// TwinCAT 3 PLC project EtherCAT_Test_1
// ProgramVersion: 3.1.4023.0
// libraries:
//   Tc2_EtherCAT, * (Beckhoff Automation GmbH)
//   Tc2_HVAC, * (Beckhoff Automation GmbH)
//   Tc2_Standard, * (Beckhoff Automation GmbH)
//   Tc2_System, * (Beckhoff Automation GmbH)
//   Tc3_Module, * (Beckhoff Automation GmbH)
// project tree:
//   DUTs/ ST_TypeOfPositioning.TcDUT
//   GVLs/ GVL.TcGVL
//   / PlcTask.TcTTO
//   POUs/ MAIN.TcPOU, P_ProfilePositionModeTest.TcPOU, P_VelocityModeTest.TcPOU, StartUpTests.TcPOU, ST_PlcErrorStartUp.TcDUT
//   POUs/ProfilePositionMode/ FB_EnableDevice.TcPOU, Motion.TcPOU
//   POUs/VelocityMode/ BasicTests.TcPOU, VelocityMode.TcPOU

CONFIGURATION EtherCAT_Test_1
    RESOURCE PLC ON TwinCAT3
        TASK PlcTask(INTERVAL := T#10ms, PRIORITY := 20);
        PROGRAM MAIN WITH PlcTask : MAIN;
    END_RESOURCE
END_CONFIGURATION

// ---- DUTs/ST_TypeOfPositioning.TcDUT
TYPE ST_TypeOfPositioning :
STRUCT
	bStartImmediately			: BOOL; (*if Bool is true, target position is absolute, otherwise relative*)
	bAbsolutePositioning		: BOOL; (*if Bool is true, velocity does not change, when first target position is reached - no braking*)
	bChangeOnSetPoint			: BOOL; (*if set true, moving command is executed immediately*)
	nReferencing				: BYTE;
	(*describes positioning behaviour 
		- 1: Positioning relative to previous target position
		- 2: Positioning relative to default value of ramp generator
		- 3: Positioning relative to actual position*)	
END_STRUCT
END_TYPE

// ---- POUs/ST_PlcErrorStartUp.TcDUT
TYPE ST_PlcErrorStartUp :
STRUCT
	bPlcError		: BOOL;
	bErrorCode		: ARRAY[1..4] OF UDINT;
END_STRUCT
END_TYPE

// ---- GVLs/GVL.TcGVL
{attribute 'qualified_only'}
VAR_GLOBAL
	sNetId				: T_AmsNetId := '5.109.65.175.2.1';
	nSlaveAddr			: UINT := 1004;
	
	Controlword AT%Q*		: UINT;	
	Statusword AT%I*		: UINT;
	
	bReset					: BOOL;
END_VAR

// ---- POUs/MAIN.TcPOU
PROGRAM MAIN
VAR_INPUT
	Controlword AT%Q*		: UINT;	
	TargetPosition AT%Q*	: DINT;
END_VAR
VAR_OUTPUT
	Statusword AT%I*		: UINT;
END_VAR

VAR
	bStartUpTest			: BOOL;
	bVelocityModeActive		: BOOL := FALSE;
END_VAR	

VAR
	aTemperatureObjects		: ARRAY[1..2] OF INT := [1,1]; 	//0x2200, 0x2202
	aMOPObjects				: ARRAY[1..2] OF INT := [1,1]; 	//0x6060, 0x6061
	aControlStatusWords		: ARRAY[1..2] OF INT := [1,1]; 	//0x6040, 0x6041
	bTargetPosition			: BOOL;							//0x607A
	
	fbSetToPPMode			: FB_EcCoeSdoWrite;
	fbSetToVelocityMode		: FB_EcCoeSdoWrite;
	bSetToPPMode			: BOOL;
	bSetToVelocityMode		: BOOL := TRUE;
	tSetToPPMode			: TON;
	fSetToVelocityMode		: F_TRIG;
	nModeOfOperation		: UDINT := 2;
	bBasicTest 				: BOOL := FALSE;
END_VAR

//StartUpTests(bTrigger := bStartUpTest,
//	aTemperatureObjects := aTemperatureObjects,
//	aControlStatusWords := aControlStatusWords,
//	aMOPObjects := aMOPObjects,
//	sNetID := GVL.sNetId,
//	nSlaveAddr := GVL.nSlaveAddr);
(*
fbSetToPPMode(sNetId := GVL.sNetId, 
				nSlaveAddr := GVL.nSlaveAddr,
				nIndex := 16#6060,
				pSrcBuf := ADR(nModeOfOperation),
				cbBufLen := SIZEOF (nModeOfOperation),
				bExecute := bSetToPPMode);
tSetToPPMode(IN := bSetToPPMode,
				PT := T#250MS);
bSetToPPMode := TRUE;
IF tSetToPPMode.Q THEN
	P_ProfilePositionModeTest();	
END_IF
*)
IF bBasicTest THEN
	BasicTests();
ELSE
//TODO read IF velocitymode was set via FB
fbSetToVelocityMode(sNetId := GVL.sNetId, 
				nSlaveAddr := GVL.nSlaveAddr,
				nIndex := 16#6060,
				pSrcBuf := ADR(nModeOfOperation),
				cbBufLen := SIZEOF (nModeOfOperation),
				bExecute := bSetToVelocityMode);
fSetToVelocityMode(CLK := fbSetToVelocityMode.bBusy);

IF fSetToVelocityMode.Q THEN
	bVelocityModeActive := TRUE;
	ADSLOGSTR(msgCtrlMask := ADSLOG_MSGTYPE_HINT,
				msgFmtStr := 'Set to velocity mode.',
				strArg := '');
END_IF
IF bVelocityModeActive THEN
	P_VelocityModeTest();
END_IF
END_IF

END_PROGRAM

// ---- POUs/VelocityMode/BasicTests.TcPOU
PROGRAM BasicTests
VAR
	bSetVelocity			: BOOL;
	bStop					: BOOL;
	nTargetVelocity 		: DINT := 1000;
	fbGetStatusword			: FB_EcCoeSdoRead;
	fbSetVelocityWindow 	: FB_EcCoeSdoWrite;
	fbSetVelocityWindowTime	: FB_EcCoeSdoWrite;
	fbProfileVelocityMode 	: ProfileVelocityMode;
	nStatusWord				: DINT;
	bGetStatusword			: BOOL;
	tGetStatusword: TON;
	bTargetReached: BOOL;
	bSpeedIsZero: BOOL;
	nVelocityWindow		: DINT := 50;
	bSetVelocityWindow: BOOL;
	nVelocityWindowTime: DINT := 100;
END_VAR


fbProfileVelocityMode(sNetID := GVL.sNetId,
					nSlaveAddr := GVL.nSlaveAddr,
					nTargetVelocity := nTargetVelocity,
					bSetVelocity := bSetVelocity);	
			
IF bStop THEN
	MAIN.Controlword := 0;
	GVL.bReset := TRUE;
	bStop := FALSE;
END_IF

tGetStatusword(IN := bGetStatusword,
					PT := T#50MS);	
IF tGetStatusword.Q THEN
	bGetStatusword := FALSE;
ELSE
	bGetStatusword := TRUE;		
END_IF
// set parameter
fbSetVelocityWindow(sNetId := GVL.sNetId,
						nSlaveAddr := GVL.nSlaveAddr,
						nIndex := 16#606D,
						nSubindex := 0,
						pSrcBuf := ADR(nVelocityWindow),
						cbBufLen := SIZEOF(nVelocityWindow),
						bExecute := bSetVelocityWindow);
fbSetVelocityWindow(sNetId := GVL.sNetId,
						nSlaveAddr := GVL.nSlaveAddr,
						nIndex := 16#606F,
						nSubindex := 0,
						pSrcBuf := ADR(nVelocityWindow),
						cbBufLen := SIZEOF(nVelocityWindow),
						bExecute := bSetVelocityWindow);
						
fbSetVelocityWindowTime(sNetId := GVL.sNetId,
						nSlaveAddr := GVL.nSlaveAddr,
						nIndex := 16#606E,
						nSubindex := 0,
						pSrcBuf := ADR(nVelocityWindowTime),
						cbBufLen := SIZEOF(nVelocityWindowTime),
						bExecute := bSetVelocityWindow);
fbSetVelocityWindowTime(sNetId := GVL.sNetId,
						nSlaveAddr := GVL.nSlaveAddr,
						nIndex := 16#6070,
						nSubindex := 0,
						pSrcBuf := ADR(nVelocityWindowTime),
						cbBufLen := SIZEOF(nVelocityWindowTime),
						bExecute := bSetVelocityWindow);
//end set parameters

fbGetStatusword(sNetId := GVL.sNetId,
				nSlaveAddr := GVL.nSlaveAddr,
				nIndex := 16#6041,
				nSubindex := 0,
				pDstBuf := ADR(nStatusWord),
				cbBufLen := SIZEOF(nStatusWord),
				bExecute := bGetStatusword);
				
IF nStatusWord.10 THEN
	bTargetReached := TRUE;
ELSE
	bTargetReached := FALSE;
END_IF				
IF nStatusWord.12 THEN
	bSpeedIsZero := TRUE;
ELSE
	bSpeedIsZero := FALSE;
END_IF

END_PROGRAM

// ---- POUs/P_VelocityModeTest.TcPOU
PROGRAM P_VelocityModeTest
//general handling
VAR
	bStartTestOfNewDrive			: BOOL;//starts new test
	bRestartTest					: BOOL;//restart if single test failed
	bManuallyRestoreDefaultValues	: BOOL;
	bError							: BOOL := FALSE;//Error handling
	bAckError						: BOOL;//Error handling
	bStopMotor						: BOOL;//Error handling
	bOnFirstIn						: BOOL := TRUE;
END_VAR

//test case success indication variables
VAR
	bSingleTestFailed					: BOOL := FALSE;
	
	bObject6042tested				: BOOL := FALSE;//test case success indication variables
	bObject6043tested				: BOOL := FALSE;//test case success indication variables
	bObject6046tested				: BOOL := FALSE;//test case success indication variables
	bObject6048tested				: BOOL := FALSE;//test case success indication variables
	bObject6049tested				: BOOL := FALSE;//test case success indication variables
	
	bTestBasicOperation_Success		: BOOL := FALSE;//test case success indication variables
	bTestAccel_Success				: BOOL := FALSE;//test case success indication variables	
	bTestDecel_Success				: BOOL := FALSE;//test case success indication variables
	bTestLimits_Success				: BOOL := FALSE;//test case success indication variables
	
	bTestBasicOperation_Failed		: BOOL := FALSE;
	bTestAccel_Failed				: BOOL := FALSE;
	bTestDecel_Failed				: BOOL := FALSE;
	bTestLimits_Failed				: BOOL := FALSE;
	
	bMaxLimitTest_Success			: BOOL := FALSE; //helper for limit
	bMinLimitTest_Success			: BOOL := FALSE; //helper for limit
	bMaxLimitTest_Failed			: BOOL := FALSE; //helper for limit
	bMinLimitTest_Failed			: BOOL := FALSE; //helper for limit	
END_VAR

//relevant parameters for test options
VAR
	fToleranceLimit					: REAL := 0.2; // 20% tolerance
	fToleranceAccDec				: REAL := 0.1; // 10% tolerance
	fToleranceBasicOp				: REAL := 0.02; // 2% tolerance
	nDeltaSpeedRef					: DINT := 300; //speed reference for acc/dec
	nDeltaTimeRef					: DINT := 1; //time reference for acc/dec
	nMinLimitRef					: DINT := 200; //testing this minimum velocity limit
	nMaxLimitRef					: DINT := 1000; //testing this maximum velocity limit	
END_VAR

// default values will be deliberately changed. Persistent variables keep their values also at shutdown of PLC, see https://infosys.beckhoff.com/index.php?content=../content/1031/tc3_plc_intro/2526557579.html&id=
// pressing "restart in run modus" will NOT clear these values!
VAR PERSISTENT
	nDefaultAccSpeed				: DINT;
	nDefaultDecSpeed				: DINT;
	nDefaultAccTime					: DINT;
	nDefaultDecTime					: DINT;
	nDefaultVelocityMinLimit		: DINT;
	nDefaultVelocityMaxLimit		: DINT;
END_VAR

// all variables
VAR	
	eTestMode	: (WAIT_FOR_TEST, READ_DEFAULT_VALUES, WRITE_DEFAULT_VALUES, ERROR, STOP_DRIVE, BASIC_OPERATION, TEST_ACCEL, TEST_DECEL, TEST_LIMITS); 
	step							: INT := 1;
	stepTestMode					: INT := 0; //start in idle mode
	
	bSetControlWord					: BOOL := TRUE;
	fbVelocityMode					: VelocityMode;
	fbGetStatusword					: FB_EcCoeSdoRead;
	fbGetActualVelocity				: FB_EcCoeSdoRead;
//	fbGetVelocityLimitMax			: FB_EcCoeSdoRead;
//	fbGetVelocityLimitMin			: FB_EcCoeSdoRead;
	fbReadVelocityLimits1			: FB_EcCoeSdoRead;
	fbReadVelocityLimits2			: FB_EcCoeSdoRead;
	fbWriteVelocityLimits1			: FB_EcCoESdoWrite;
	fbWriteVelocityLimits2			: FB_EcCoESdoWrite;
	fbWriteAcc1						: FB_EcCoESdoWrite;
	fbWriteAcc2						: FB_EcCoESdoWrite;
	fbReadAcc1						: FB_EcCoeSdoRead;
	fbReadAcc2						: FB_EcCoeSdoRead;
	fbWriteDec1						: FB_EcCoESdoWrite;
	fbWriteDec2						: FB_EcCoESdoWrite;
	fbReadDec1						: FB_EcCoeSdoRead;
	fbReadDec2						: FB_EcCoeSdoRead;
	fbGetVelocityDemand				: FB_EcCoESdoRead;
	fbGetTargetVelocity				: FB_EcCoESdoRead;
	nTargetVelocity					: DINT := 50; //rpm
	nActualVelocity					: DINT;
	nStatusword						: UINT;
	nSpeed							: DINT;
	nTime							: DINT;
		
	bGetCurrentVelocity				: BOOL;
	bGetStatusword					: BOOL;
	bSetVelocity					: BOOL; 
	nTargetVelocityAfterLimit		: DINT;
	tTimeDec1						: TIME;
	tTimeDec2						: TIME;
	nAccMeasured					: REAL;
	nDecMeasured					: REAL;
	bIsAccelerating					: BOOL;
	bIsDecelerating					: BOOL;
	
	bDone							: BOOL;
	nDeltaVelocityTarget			: REAL;
	fDesiredAcceleration			: REAL;
	nVelocityDemand					: DINT;
	nVelocityMinLimit 				: DINT;
	nVelocityMaxLimit 				: DINT;
	bWriteDefaultValues				: BOOL;
	nDecVelocity					: DINT;
	fDesiredDeceleration			: REAL;
	bStopAfterLimitTest				: BOOL;

	tTimeout						: TON;
	tTimer							: TON;
	tGetStatusword					: TON;
	tWaitForCurrentVelocity			: TON;
	tTimeAcc1						: TIME;
	tTimeAcc2						: TIME;
	tDiff							: TIME;
	fTrigger						: F_TRIG;
	fFlag 							: F_TRIG;
	fFlag2 							: F_TRIG;	
	ShowLimitVelocity				: DINT;
END_VAR

IF bTestBasicOperation_Failed OR bTestAccel_Failed OR bTestDecel_Failed OR bMinLimitTest_Failed OR bMaxLimitTest_Failed OR bTestLimits_Failed THEN
	bSingleTestFailed := TRUE;
ELSE bSingleTestFailed := FALSE;
END_IF


tWaitForCurrentVelocity(IN := bGetCurrentVelocity,
							PT := T#10MS);
tGetStatusword(IN := bGetStatusword,
					PT := T#500MS);	
							
IF tWaitForCurrentVelocity.Q THEN
	bGetCurrentVelocity := FALSE;
ELSE
	bGetCurrentVelocity := TRUE;		
END_IF
// read FBs
fbGetStatusword(sNetId := GVL.sNetId,
				nSlaveAddr := GVL.nSlaveAddr,
				nIndex := 16#6041,
				nSubindex := 0,
				pDstBuf := ADR(nStatusWord),
				cbBufLen := SIZEOF(nStatusWord),
				bExecute := bGetStatusword);
				
fbGetActualVelocity(sNetId := GVL.sNetId,
					nSlaveAddr := GVL.nSlaveAddr,
					nIndex := 16#6044,
					nSubindex := 0,
					pDstBuf := ADR(nActualVelocity),
					cbBufLen := SIZEOF(nActualVelocity),
					bExecute := bGetCurrentVelocity);

//write to motor
MAIN.Controlword.4 := bSetControlWord; //velocity demand value shall equal to ramp output value
MAIN.Controlword.5 := bSetControlWord; //ramp output value shall follow ramp input value
MAIN.Controlword.6 := bSetControlWord; //ramp input value shall accord with ramp reference

			
//stop
IF bStopMotor THEN
	MAIN.Controlword := 0;
	stepTestMode := 0;
END_IF


(*TEST SUITE*)	
//error detection
IF bError THEN
	MAIN.Controlword := 0;
	stepTestMode := 0;
	eTestMode := ERROR;
END_IF
// restore stored default values
IF bManuallyRestoreDefaultValues THEN
	bError := FALSE;
	stepTestMode := 0;
	eTestMode := WRITE_DEFAULT_VALUES;
END_IF

CASE eTestMode OF
	WAIT_FOR_TEST:
		tTimeout(IN := FALSE);
		step := 1; //resetting general step counter for use within TestModes
		CASE stepTestMode OF
			0: //idle
				IF bRestartTest THEN //restart inside a test procedure
					GVL.bReset := TRUE;
					bRestartTest := FALSE; 
					bSetControlWord := TRUE;
					bTestBasicOperation_Failed := bTestAccel_Failed := bTestDecel_Failed := bMinLimitTest_Failed := bMaxLimitTest_Failed := bTestLimits_Failed := FALSE;
					stepTestMode := stepTestMode+1;
				END_IF
				IF bStartTestOfNewDrive THEN //start test of a new drive 
					GVL.bReset := TRUE;
					Reset();
					bSetControlWord := TRUE;
					bStartTestOfNewDrive := FALSE;
					eTestMode := READ_DEFAULT_VALUES;
				END_IF
		
			1: 
				IF bTestBasicOperation_Success THEN 
					stepTestMode := stepTestMode+1; 
					bObject6043tested := TRUE;
				ELSE 
					eTestMode := BASIC_OPERATION; 
					ADSLOGSTR(msgCtrlMask := ADSLOG_MSGTYPE_HINT, msgFmtStr := 'Testing basic operation...', strArg := '');
				END_IF 				
			2: 				
				IF bTestAccel_Success THEN 
					stepTestMode := stepTestMode+1; 
					bObject6048tested := TRUE;
				ELSIF nActualVelocity = 0 THEN 
					eTestMode := TEST_ACCEL; 
					bSetControlWord := TRUE; 
					ADSLOGSTR(msgCtrlMask := ADSLOG_MSGTYPE_HINT, msgFmtStr := 'Testing acceleration...', strArg := '');
				END_IF 				
			3: 
				IF bTestDecel_Success THEN 
					stepTestMode := stepTestMode+1; 
					bObject6049tested := TRUE;
				ELSE 
					eTestMode := TEST_DECEL; 
					ADSLOGSTR(msgCtrlMask := ADSLOG_MSGTYPE_HINT, msgFmtStr := 'Testing deceleration...', strArg := '');
				END_IF
			4: 
				IF bTestLimits_Success THEN 
					stepTestMode := stepTestMode+1; 
					bObject6046tested := TRUE;
				ELSE 
					eTestMode := TEST_LIMITS; 
					ADSLOGSTR(msgCtrlMask := ADSLOG_MSGTYPE_HINT, msgFmtStr := 'Testing limits...', strArg := '');
				END_IF				
			
			5: //all tests successful
				MAIN.Controlword := 0;
				ADSLOGSTR(msgCtrlMask := ADSLOG_MSGTYPE_HINT, msgFmtStr := 'All tests successful!', strArg := '');
				stepTestMode := 0; //idle
		END_CASE	
	
		
	(* Error handling *)
	ERROR:
		MAIN.Controlword := 0;
		bSetControlWord := FALSE;
		step := 1;
		IF bAckError OR bRestartTest THEN
			bAckError := FALSE;
			bError := FALSE;
			
			eTestMode := WAIT_FOR_TEST;
			stepTestMode := 0;
		END_IF


	READ_DEFAULT_VALUES: 
		CASE step OF
			1: //read acc
				ReadAcc(nDeltaSpeed := nDefaultAccSpeed, nDeltaTime := nDefaultAccTime, bDone => bDone);
				IF bDone THEN
					step := step+1;
				END_IF
			2: //read dec
				ReadDec(nDeltaSpeed := nDefaultDecSpeed, nDeltaTime := nDefaultDecTime, bDone => bDone);
				IF bDone THEN
					step := step+1;
				END_IF				
			3: //read limits
				ReadVelocityLimits(nVelocityMinLimit := nDefaultVelocityMinLimit, nVelocityMaxLimit := nDefaultVelocityMaxLimit, bDone => bDone);
				IF bDone THEN
					step := step+1;
				END_IF
			4: 
				eTestMode := WAIT_FOR_TEST;			
				ADSLOGSTR(msgCtrlMask := ADSLOG_MSGTYPE_HINT, msgFmtStr := 'Default values read.', strArg := '');
				stepTestMode := 1; //start test basic operation
		END_CASE
		
		
	WRITE_DEFAULT_VALUES: 
		IF bOnFirstIn THEN 
			step := 1;
		END_IF
		CASE step OF
			1: //write acc
				bOnFirstIn := FALSE;
				WriteAcc(nDeltaSpeedRef := nDefaultAccSpeed, nDeltaTimeRef := nDefaultAccTime, bDone => bDone);
				IF bDone THEN
					step := step+1;
				END_IF
			2: 
				ReadAcc(nDeltaSpeed := nSpeed, nDeltaTime := nTime, bDone => bDone);
				IF nSpeed = nDefaultAccSpeed AND nTime = nDefaultAccTime AND bDone THEN
					step := step+1;
				END_IF
			3: //write dec
				WriteDec(nDeltaSpeedRef := nDefaultDecSpeed, nDeltaTimeRef := nDefaultDecTime, bDone => bDone);
				IF bDone THEN
					step := step+1;
				END_IF	
			4:
				ReadDec(nDeltaSpeed := nSpeed, nDeltaTime := nTime, bDone => bDone);
				IF nSpeed = nDefaultDecSpeed AND nTime = nDefaultDecTime AND bDone THEN
					step := step+1;
				END_IF
			
			5: //write limits
				WriteVelocityLimits(nVelocityMinLimit := nDefaultVelocityMinLimit, nVelocityMaxLimit := nDefaultVelocityMaxLimit, bDone => bDone);
				IF bDone THEN
					step := step+1;
				END_IF
			6: 
				ReadVelocityLimits(nVelocityMinLimit := nVelocityMinLimit, nVelocityMaxLimit := nVelocityMaxLimit, bDone => bDone);
				IF nVelocityMinLimit = nDefaultVelocityMinLimit AND nVelocityMaxLimit = nDefaultVelocityMaxLimit AND bDone THEN
					step := step+1;
				END_IF

			7: 
				eTestMode := WAIT_FOR_TEST;	
				ADSLOGSTR(msgCtrlMask := ADSLOG_MSGTYPE_HINT,
					msgFmtStr := 'Default values restored. Acc, dec and limits',
					strArg := '');		
				IF bSingleTestFailed THEN
					bError := TRUE;
				END_IF
				IF bStopAfterLimitTest THEN
					bStopAfterLimitTest := FALSE;
					eTestMode := STOP_DRIVE;
				END_IF
				bManuallyRestoreDefaultValues := FALSE;
				bOnFirstIn := TRUE;
		END_CASE
		
		
	STOP_DRIVE:
		step := 1;
		nTargetVelocity := 0;
		tTimeout(IN := TRUE, PT := T#15S);
		bSetVelocity := TRUE;
		fbVelocityMode(sNetID := GVL.sNetId,
					nSlaveAddr := GVL.nSlaveAddr,
					nTargetVelocity := nTargetVelocity,
					bSetVelocity := bSetVelocity,
					nTargetVelocityAfterLimit => nTargetVelocityAfterLimit);
		IF nActualVelocity = 0 THEN
			IF bWriteDefaultValues THEN
				bWriteDefaultValues := FALSE;
				eTestMode := WRITE_DEFAULT_VALUES;
			ELSE
				eTestMode := WAIT_FOR_TEST;
			END_IF
		END_IF
		
		IF tTimeout.Q THEN
			bError := TRUE;
			ADSLOGSTR(msgCtrlMask := ADSLOG_MSGTYPE_HINT,
				msgFmtStr := 'Timeout when shutting down drive. Please restore default values manually.',
				strArg := '');
		END_IF
	
	(* Test basic operation *)
	BASIC_OPERATION:
		tTimeout(IN := TRUE, PT := T#10S);
		CASE step OF
		1:	
			nTargetVelocity := 300; //rpm
			bSetVelocity := TRUE;
			fbVelocityMode(sNetID := GVL.sNetId,
						nSlaveAddr := GVL.nSlaveAddr,
						nTargetVelocity := nTargetVelocity,
						bSetVelocity := bSetVelocity,
						nTargetVelocityAfterLimit => nTargetVelocityAfterLimit);
			IF NOT fbVelocityMode.bBusy THEN //now velocity is set
				step := step+1;
			END_IF				
		2: 
			fbGetTargetVelocity(sNetId := GVL.sNetId,
				nSlaveAddr := GVL.nSlaveAddr,
				nIndex := 16#6042,
				nSubIndex := 0,
				pDstBuf := ADR(nVelocityDemand),
				cbBufLen := SIZEOF(nVelocityDemand),
				bExecute := TRUE);
			fFlag(CLK := fbGetTargetVelocity.bBusy);
			IF fFlag.Q AND nVelocityDemand = nTargetVelocity THEN
				fbGetTargetVelocity(bExecute := FALSE);
				bObject6042tested := TRUE;
				step := step+1;
			END_IF		
		3:  
			tTimer(IN:=TRUE, PT:=T#3S);
			IF tTimer.Q THEN
				tTimer(IN:=FALSE);
				step := step+1;
			END_IF
		4:
			IF  TO_REAL(nActualVelocity) > ((1-fToleranceBasicOp)*TO_REAL(nTargetVelocityAfterLimit)) 
			AND TO_REAL(nActualVelocity) < ((1+fToleranceBasicOp)*TO_REAL(nTargetVelocityAfterLimit)) THEN // Vsoll = Vist with 2% tolerance
				fbGetVelocityDemand(sNetId := GVL.sNetId,
					nSlaveAddr := GVL.nSlaveAddr,
					nIndex := 16#6043,
					nSubIndex := 0,
					pDstBuf := ADR(nVelocityDemand),
					cbBufLen := SIZEOF(nVelocityDemand),
					bExecute := TRUE);
				fFlag2(CLK := fbGetVelocityDemand.bBusy);
				
				IF fFlag2.Q THEN
					fbGetVelocityDemand(bExecute := FALSE);
					IF nVelocityDemand = nTargetVelocity THEN
						bTestBasicOperation_Success := TRUE; //set success indication	
						step := step+1;								
						ADSLOGSTR(msgCtrlMask := ADSLOG_MSGTYPE_HINT,
							msgFmtStr := 'Basic operation test success.',
							strArg := '');
					END_IF
				END_IF
			ELSIF nActualVelocity > 2*nTargetVelocityAfterLimit THEN
				bError := TRUE;
				bTestBasicOperation_Failed := TRUE;
			END_IF				
			
		5:	//soft stop motor
			eTestMode := STOP_DRIVE;			
		END_CASE
		
		//Error handling in wait_for_test
		IF tTimeout.Q THEN
			bTestBasicOperation_Failed := TRUE;
			bError := TRUE;
			ADSLOGSTR(msgCtrlMask := ADSLOG_MSGTYPE_HINT,
				msgFmtStr := 'Basic operation test failed. Timeout.',
				strArg := '');
		END_IF

	
	(* Test acceleration target *)
	TEST_ACCEL:
		tTimeout(IN := TRUE, PT := T#10S); 
		CASE step OF
			1: //set acceleration values
				WriteAcc(nDeltaSpeedRef := nDeltaSpeedRef, nDeltaTimeRef := nDeltaTimeRef, bDone => bDone);
				IF bDone THEN
					step := step+1;
				END_IF
				
			2: //read acceleration
				ReadAcc(nDeltaSpeed := nSpeed, nDeltaTime := nTime, bDone => bDone); 
				IF nSpeed = nDeltaSpeedRef AND nTime = nDeltaTimeRef AND bDone THEN //Acceleration values were set correctly
					step := step+1;
				END_IF
				
			3: //set drive to TargetVelocity and measure acceleration time
				nTargetVelocity := 2000;
				nDeltaVelocityTarget := 0.995*TO_REAL(nTargetVelocity); //needs to be a little lower than target due to acc ramping
				fDesiredAcceleration := TO_REAL(nDeltaSpeedRef/nDeltaTimeRef); // acc reference
				
				bSetVelocity := TRUE;
				fbVelocityMode(sNetID := GVL.sNetId,
							nSlaveAddr := GVL.nSlaveAddr,
							nTargetVelocity := nTargetVelocity,
							bSetVelocity := bSetVelocity,
							nTargetVelocityAfterLimit => nTargetVelocityAfterLimit);
				fTrigger(CLK := fbVelocityMode.bBusy);
				IF fTrigger.Q THEN
					tTimeAcc1 := TIME();
					step := step+1;
				END_IF
			
			4:
				tTimer(IN:=TRUE, PT:=T#50MS);
				IF tTimer.Q THEN
					tTimer(IN:=FALSE);
					step := step+1;
				END_IF
				
			5:
				IF TO_REAL(nActualVelocity) >= nDeltaVelocityTarget THEN 
					tTimeAcc2 := TIME();
					tDiff := tTimeAcc2 - tTimeAcc1; //time difference of drive to reach nSpeedRef
					nAccMeasured := TO_REAL(nActualVelocity*1000/TIME_TO_DINT(tDiff)); //time in ms
					step := step+1;
				END_IF

			6: //validate result
				IF  nAccMeasured > ((1-fToleranceAccDec)*fDesiredAcceleration) 
				AND nAccMeasured < ((1+fToleranceAccDec)*fDesiredAcceleration) THEN //within range of tolerance: default 10%
					bTestAccel_Success := TRUE;
					ADSLOGSTR(msgCtrlMask := ADSLOG_MSGTYPE_HINT,
					msgFmtStr := 'Acceleration test success.',
					strArg := '');
				ELSE
					bTestAccel_Failed := TRUE;
					ADSLOGSTR(msgCtrlMask := ADSLOG_MSGTYPE_HINT,
						msgFmtStr := 'Acceleration test failed. Motor acceleration not within range of reference values.',
						strArg := '');
				END_IF
				bWriteDefaultValues := TRUE;
				eTestMode := STOP_DRIVE; //stop and restore default variables
		END_CASE
		
		//Error handling timeout
		IF tTimeout.Q THEN
			eTestMode := WRITE_DEFAULT_VALUES; //restore default variables
			bTestAccel_Failed := TRUE;
			ADSLOGSTR(msgCtrlMask := ADSLOG_MSGTYPE_HINT,
				msgFmtStr := 'Acceleration test failed. Timeout.',
				strArg := '');
		END_IF
		
	
		
(* Test acceleration target *)
	TEST_DECEL:
		tTimeout(IN := TRUE, PT := T#15S); 
		CASE step OF
			1: //set deceleration values
				WriteDec(nDeltaSpeedRef := nDeltaSpeedRef, nDeltaTimeRef := nDeltaTimeRef, bDone => bDone);
				IF bDone THEN
					step := step+1;
				END_IF
				
			2: //read deceleration
				ReadDec(nDeltaSpeed := nSpeed, nDeltaTime := nTime, bDone => bDone); 
				IF nSpeed = nDeltaSpeedRef AND nTime = nDeltaTimeRef AND bDone THEN //Acceleration values were set correctly
					step := step+1;
				END_IF
				
			3: //set drive to velocity
				nTargetVelocity := 1500;
				nDecVelocity := nTargetVelocity;	
				fDesiredDeceleration := TO_REAL(nDeltaSpeedRef/nDeltaTimeRef); // dec reference		
				bSetVelocity := TRUE;
				fbVelocityMode(sNetID := GVL.sNetId,
							nSlaveAddr := GVL.nSlaveAddr,
							nTargetVelocity := nTargetVelocity,
							bSetVelocity := bSetVelocity,
							nTargetVelocityAfterLimit => nTargetVelocityAfterLimit);
				tTimer(IN:=TRUE, PT:=T#1500MS);
				IF tTimer.Q THEN
					tTimer(IN:=FALSE);
					step := step+1;
				END_IF
			
			4:
				IF nActualVelocity > 0.99*nTargetVelocityAfterLimit THEN 
					nTargetVelocity := 0;
					step := step+1;
				END_IF

			5: //test run of drive for validation of deceleration 
				bSetVelocity := TRUE;
				fbVelocityMode(sNetID := GVL.sNetId,
							nSlaveAddr := GVL.nSlaveAddr,
							nTargetVelocity := nTargetVelocity,
							bSetVelocity := bSetVelocity,
							nTargetVelocityAfterLimit => nTargetVelocityAfterLimit);
				fTrigger(CLK := fbVelocityMode.bBusy);
				IF fTrigger.Q THEN
					tTimeDec1 := TIME();
					step := step+1;
				END_IF
				
			6:
				IF nActualVelocity = nTargetVelocity THEN
					tTimeDec2 := TIME();
					tDiff := tTimeDec2 - tTimeDec1; //time difference of drive to decelerate
					nDecMeasured := TO_REAL(nDecVelocity*1000/TIME_TO_DINT(tDiff));
					step := step+1;
				END_IF
			
			7:	//validation
				IF  nDecMeasured > ((1-fToleranceAccDec)*fDesiredDeceleration) 
				AND nDecMeasured < ((1+fToleranceAccDec)*fDesiredDeceleration) THEN //within range of tolerance: default 10%
					bTestDecel_Success := TRUE;
					ADSLOGSTR(msgCtrlMask := ADSLOG_MSGTYPE_HINT,
					msgFmtStr := 'Deceleration test success.',
					strArg := '');
				ELSE
					bTestDecel_Failed := TRUE;
					ADSLOGSTR(msgCtrlMask := ADSLOG_MSGTYPE_WARN,
						msgFmtStr := 'Deceleration test failed. Motor deceleration not within range of reference values.',
						strArg := '');
				END_IF
				bWriteDefaultValues := TRUE;
				eTestMode := STOP_DRIVE; //stop and restore default variables
		END_CASE
		
		//Error handling timeout
		IF tTimeout.Q THEN
			eTestMode := WRITE_DEFAULT_VALUES; //restore default variables
			bTestDecel_Failed := TRUE;
			ADSLOGSTR(msgCtrlMask := ADSLOG_MSGTYPE_WARN,
				msgFmtStr := 'Deceleration test failed. Timeout.',
				strArg := '');
		END_IF
		

	
//	(* Test velocity limtis *)
	TEST_LIMITS: 
		tTimeout(IN:=TRUE, PT:=T#15S);
		CASE step OF
			1: 
				nTargetVelocity := 2000;
				WriteVelocityLimits(nVelocityMinLimit := nMinLimitRef, nVelocityMaxLimit := nMaxLimitRef, bDone => bDone);
				IF bDone THEN
					step := step+1;
				END_IF
				
			2: //test max limit
				bSetVelocity := TRUE;
				fbVelocityMode(sNetID := GVL.sNetId,
							nSlaveAddr := GVL.nSlaveAddr,
							nTargetVelocity := nTargetVelocity,
							bSetVelocity := bSetVelocity,
							nTargetVelocityAfterLimit => nTargetVelocityAfterLimit);
				IF NOT fbVelocityMode.bBusy THEN
					bIsAccelerating := TRUE;
					step := step+1;
				END_IF
			
			3:
				tTimer(IN := bIsAccelerating, PT := T#3S); //run for x seconds
				IF tTimer.Q THEN 
					tTimer(IN:=FALSE);
					step := step+1;
				END_IF
			
			4:
				IF TO_REAL(nActualVelocity) > ((1+fToleranceLimit)*TO_REAL(nMaxLimitRef))(* 20% overshot accounted *) THEN 
					bMaxLimitTest_Failed := TRUE;
					eTestMode := WRITE_DEFAULT_VALUES;
					ADSLOGSTR(msgCtrlMask := ADSLOG_MSGTYPE_WARN,
						msgFmtStr := 'Max limit test failed.',
						strArg := '');			
				ELSE
					bMaxLimitTest_Success := TRUE;
					ADSLOGSTR(msgCtrlMask := ADSLOG_MSGTYPE_HINT,
						msgFmtStr := 'Max limit test success.',
						strArg := '');
					step := step+1;
				END_IF
				bIsAccelerating := FALSE;
				nTargetVelocity := 0;
				
			5: //test min limit
				bSetVelocity := TRUE;
				fbVelocityMode(sNetID := GVL.sNetId,
							nSlaveAddr := GVL.nSlaveAddr,
							nTargetVelocity := nTargetVelocity,
							bSetVelocity := bSetVelocity,
							nTargetVelocityAfterLimit => nTargetVelocityAfterLimit);
				IF NOT fbVelocityMode.bBusy THEN
					bIsDecelerating := TRUE;
					step := step+1;
				END_IF
								
			6:
				tTimer(IN := bIsDecelerating, PT := T#3S); //run for x seconds
				IF tTimer.Q THEN 
					tTimer(IN:=FALSE);
					step := step+1;
				END_IF
			
			7:
				// a way for dynamic time determination
//				fTimeFaktor := DINT_TO_REAL((nActualVelocity-nTargetVelocity)/nSpeedDec); 
//				tDecTime := REAL_TO_TIME(2000+fTimeFaktor * nDefaultDecTime*1000); //acceleration time, min 2s
//				tTimer(IN := bIsDecelerating, PT := tDecTime);
				IF TO_REAL(nActualVelocity) < ((1-fToleranceLimit)*TO_REAL(nMinLimitRef))(*20% overshot accounted*) THEN 
					bMinLimitTest_Failed := TRUE;
					ADSLOGSTR(msgCtrlMask := ADSLOG_MSGTYPE_WARN,
						msgFmtStr := 'Min limit test failed.',
						strArg := '');										
				ELSE //time at witch the drive would be on targetvelocity without limit acitve
					bMinLimitTest_Success := TRUE;
					ADSLOGSTR(msgCtrlMask := ADSLOG_MSGTYPE_HINT,
						msgFmtStr := 'Min limit test success.',
						strArg := '');
				END_IF
				ShowLimitVelocity := nActualVelocity;
				step := step+1;
				bIsDecelerating := FALSE;
			
			8:
				IF bMinLimitTest_Success AND bMaxLimitTest_Success THEN
					bTestLimits_Success := TRUE;
					ADSLOGSTR(msgCtrlMask := ADSLOG_MSGTYPE_HINT,
						msgFmtStr := 'Limit test success.',
						strArg := '');
				ELSE
					bTestLimits_Failed := TRUE;
				END_IF
				bStopAfterLimitTest := TRUE;
				eTestMode := WRITE_DEFAULT_VALUES; //stop and restore default variables				
		END_CASE

END_CASE

METHOD ReadAcc : BOOL
VAR_IN_OUT
	nDeltaSpeed 	: DINT;
	nDeltaTime 		: DINT;
	//bRead : BOOL;
END_VAR
VAR_OUTPUT
	bDone			: BOOL;
END_VAR
bDone := FALSE;
//IF bRead THEN
	fbReadAcc1(sNetId := GVL.sNetId,
				nSlaveAddr := GVL.nSlaveAddr,
				nIndex := 16#6048,
				nSubindex := 1, //delta speed
				pDstBuf := ADR(nDeltaSpeed),
				cbBufLen := SIZEOF(nDeltaSpeed),
				bExecute := TRUE);
	
	fbReadAcc2(sNetId := GVL.sNetId,
				nSlaveAddr := GVL.nSlaveAddr,
				nIndex := 16#6048,
				nSubindex := 2, //delta time
				pDstBuf := ADR(nDeltaTime),
				cbBufLen := SIZEOF(nDeltaTime),
				bExecute := TRUE);
//END_IF
IF NOT fbReadAcc1.bBusy AND NOT fbReadAcc2.bBusy THEN
	fbReadAcc1(bExecute := FALSE); 
	fbReadAcc2(bExecute := FALSE); 
	//bRead := FALSE;
	bDone := TRUE;
END_IF
END_METHOD

METHOD ReadDec : BOOL
VAR_IN_OUT
	nDeltaSpeed 	: DINT;
	nDeltaTime 		: DINT;
END_VAR
VAR_OUTPUT
	bDone			: BOOL;
END_VAR
bDone := FALSE;
fbReadDec1(sNetId := GVL.sNetId,
			nSlaveAddr := GVL.nSlaveAddr,
			nIndex := 16#6049,
			nSubindex := 1, //delta speed
			pDstBuf := ADR(nDeltaSpeed),
			cbBufLen := SIZEOF(nDeltaSpeed),
			bExecute := TRUE);

fbReadDec2(sNetId := GVL.sNetId,
			nSlaveAddr := GVL.nSlaveAddr,
			nIndex := 16#6049,
			nSubindex := 2, //delta time
			pDstBuf := ADR(nDeltaTime),
			cbBufLen := SIZEOF(nDeltaTime),
			bExecute := TRUE);

IF NOT fbReadDec1.bBusy AND NOT fbReadDec2.bBusy THEN
	fbReadDec1(bExecute := FALSE); 
	fbReadDec2(bExecute := FALSE); 
	bDone := TRUE;
END_IF
END_METHOD

METHOD ReadVelocityLimits : BOOL
VAR_IN_OUT
	nVelocityMinLimit 	: DINT;
	nVelocityMaxLimit 	: DINT;
END_VAR
VAR_OUTPUT
	bDone			: BOOL;
END_VAR
bDone := FALSE;
	fbReadVelocityLimits1(sNetId := GVL.sNetId,
			nSlaveAddr := GVL.nSlaveAddr,
			nIndex := 16#6046,
			nSubindex := 1, //v_min
			pDstBuf := ADR(nVelocityMinLimit),
			cbBufLen := SIZEOF(nVelocityMinLimit),
			bExecute := TRUE);
	
	fbReadVelocityLimits2(sNetId := GVL.sNetId,
			nSlaveAddr := GVL.nSlaveAddr,
			nIndex := 16#6046,
			nSubindex := 2, //v_max
			pDstBuf := ADR(nVelocityMaxLimit),
			cbBufLen := SIZEOF(nVelocityMaxLimit),
			bExecute := TRUE);
			
IF NOT fbReadVelocityLimits1.bBusy AND NOT fbReadVelocityLimits2.bBusy THEN
	fbReadVelocityLimits1(bExecute := FALSE); 
	fbReadVelocityLimits2(bExecute := FALSE); 
	bDone := TRUE;
END_IF
END_METHOD

METHOD Reset : BOOL
VAR_INPUT
END_VAR
bObject6042tested				:= FALSE;
bObject6043tested				:= FALSE;
bObject6046tested				:= FALSE;
bObject6048tested				:= FALSE;
bObject6049tested				:= FALSE;

bTestBasicOperation_Success		:= FALSE;
bTestAccel_Success				:= FALSE;	
bTestDecel_Success				:= FALSE;
bTestLimits_Success				:= FALSE;

bTestBasicOperation_Failed		:= FALSE;
bTestAccel_Failed				:= FALSE;
bTestDecel_Failed				:= FALSE;
bTestLimits_Failed				:= FALSE;
bSingleTestFailed					:= FALSE;

bMaxLimitTest_Success			:= FALSE;
bMinLimitTest_Success			:= FALSE;
bMaxLimitTest_Failed			:= FALSE;
bMinLimitTest_Failed			:= FALSE;
END_METHOD

METHOD WriteAcc : BOOL
VAR_IN_OUT
	nDeltaSpeedRef	: DINT;
	nDeltaTimeRef	: DINT;
END_VAR
VAR_OUTPUT
	bDone 			: BOOL;
END_VAR
bDone := FALSE;
fbWriteAcc1(sNetId := GVL.sNetId,
		nSlaveAddr := GVL.nSlaveAddr,
		nIndex := 16#6048,
		nSubindex := 1, //delta speed
		pSrcBuf := ADR(nDeltaSpeedRef),
		cbBufLen := SIZEOF(nDeltaSpeedRef),
		bExecute := TRUE);	
			
fbWriteAcc2(sNetId := GVL.sNetId,
		nSlaveAddr := GVL.nSlaveAddr,
		nIndex := 16#6048,
		nSubindex := 2, //delta time
		pSrcBuf := ADR(nDeltaTimeRef),
		cbBufLen := SIZEOF(nDeltaTimeRef),
		bExecute := TRUE);

IF NOT fbWriteAcc1.bBusy AND NOT fbWriteAcc2.bBusy THEN
	fbWriteAcc1(bExecute := FALSE); 
	fbWriteAcc2(bExecute := FALSE); 
	bDone := TRUE;
END_IF
END_METHOD

METHOD WriteDec : BOOL
VAR_IN_OUT
	nDeltaSpeedRef	: DINT;
	nDeltaTimeRef	: DINT;
END_VAR
VAR_OUTPUT
	bDone 			: BOOL;
END_VAR
bDone := FALSE;
fbWriteDec1(sNetId := GVL.sNetId,
		nSlaveAddr := GVL.nSlaveAddr,
		nIndex := 16#6049,
		nSubindex := 1, //delta speed
		pSrcBuf := ADR(nDeltaSpeedRef),
		cbBufLen := SIZEOF(nDeltaSpeedRef),
		bExecute := TRUE);	
			
fbWriteDec2(sNetId := GVL.sNetId,
		nSlaveAddr := GVL.nSlaveAddr,
		nIndex := 16#6049,
		nSubindex := 2, //delta time
		pSrcBuf := ADR(nDeltaTimeRef),
		cbBufLen := SIZEOF(nDeltaTimeRef),
		bExecute := TRUE);
			
IF NOT fbWriteDec1.bBusy AND NOT fbWriteDec2.bBusy THEN
	fbWriteDec1(bExecute := FALSE); 
	fbWriteDec2(bExecute := FALSE); 
	bDone := TRUE;
END_IF
END_METHOD

METHOD WriteVelocityLimits : BOOL
VAR_IN_OUT
	nVelocityMinLimit 	: DINT;
	nVelocityMaxLimit 	: DINT;
END_VAR
VAR_OUTPUT
	bDone			: BOOL;
END_VAR
bDone := FALSE;
	fbWriteVelocityLimits1(sNetId := GVL.sNetId,
			nSlaveAddr := GVL.nSlaveAddr,
			nIndex := 16#6046,
			nSubindex := 1, //v_min
			pSrcBuf := ADR(nVelocityMinLimit),
			cbBufLen := SIZEOF(nVelocityMinLimit),
			bExecute := TRUE);
	
	fbWriteVelocityLimits2(sNetId := GVL.sNetId,
			nSlaveAddr := GVL.nSlaveAddr,
			nIndex := 16#6046,
			nSubindex := 2, //v_max
			pSrcBuf := ADR(nVelocityMaxLimit),
			cbBufLen := SIZEOF(nVelocityMaxLimit),
			bExecute := TRUE);
			
IF NOT fbWriteVelocityLimits1.bBusy AND NOT fbWriteVelocityLimits2.bBusy THEN
	fbWriteVelocityLimits1(bExecute := FALSE); 
	fbWriteVelocityLimits2(bExecute := FALSE); 
	bDone := TRUE;
END_IF
END_METHOD

END_PROGRAM

// ---- POUs/VelocityMode/VelocityMode.TcPOU
FUNCTION_BLOCK VelocityMode
VAR_INPUT
	sNetID					: T_AmsNetId;
	nSlaveAddr				: UINT;
END_VAR
VAR_OUTPUT
	bSuccess				: BOOL;
	bBusy					: BOOL;
	nTargetVelocityAfterLimit: DINT;
END_VAR
VAR_IN_OUT
	bSetVelocity			: BOOL;
	nTargetVelocity			: DINT;
END_VAR
VAR
	eMotionState			: (WAIT_FOR_TRIGGER, ENABLE_DEVICE, WAIT_FOR_NEW_VELOCITY, SET_LIMIT, SET_VELOCITY, VALIDATE_VELOCITY, ACKNOWLEDGE_VELOCITY);
	fbEnableDevice			: FB_EnableDevice;
	fbSetVelocity			: FB_EcCoeSdoWrite;
	fbGetStatusword			: FB_EcCoeSdoRead;
	fbGetVelocityLimitMin	: FB_EcCoeSdoRead;
	fbGetVelocityLimitMax	: FB_EcCoeSdoRead;
	fbGetVelocityDemand		: FB_EcCoeSdoRead;
	tWait					: TON;
	tWait2					: TON;
	nStatusword				: UINT;
	bGetStatusword			: BOOL;
	bExecuteWait			: BOOL;
	bWriteToFB				: BOOL;
	fFlag		 			: F_TRIG;
	nVelocityBuff			: DINT := 0;
	nVelocityDemand			: DINT;
	fbReadVelocityLimits1	: FB_EcCoeSdoRead;
	fbReadVelocityLimits2	: FB_EcCoeSdoRead;
	bLimitActive			: BOOL;
	nVelocityLimitMin		: DINT;
	nVelocityLimitMax		: DINT;
END_VAR

IF GVL.bReset THEN
	GVL.bReset := FALSE;
	bSuccess := FALSE;
	nVelocityBuff := 0;
	eMotionState := WAIT_FOR_TRIGGER;
END_IF

ReadLimits();
bBusy := TRUE; //FB VelocityMode is busy and the target velocity is not jet set

fbSetVelocity(sNetId := sNetID,
			nSlaveAddr := nSlaveAddr,
			nSubIndex := 0,
			nIndex := 16#6042,
			pSrcBuf := ADR(nVelocityBuff),
			cbBufLen := SIZEOF(nVelocityBuff),
			bExecute := bWriteToFB);
				
	
// state machine				
CASE eMotionState OF
	WAIT_FOR_TRIGGER:
		MAIN.Controlword := 0;
		IF bSetVelocity THEN
			ADSLOGSTR(msgCtrlMask := ADSLOG_MSGTYPE_HINT,
				msgFmtStr := 'Enable Device',
				strArg := '');
			eMotionState := ENABLE_DEVICE;
		END_IF	

	ENABLE_DEVICE:
		fbEnableDevice (bTrigger := bSetVelocity,
						bSuccess => bSuccess,
						sNetId := sNetId,
						nSlaveAddr := nSlaveAddr);
		IF fbEnableDevice.bFinished THEN
			IF NOT bSuccess THEN
				ADSLOGSTR(msgCtrlMask := ADSLOG_MSGTYPE_HINT,
					msgFmtStr := 'Device not successfully enabled',
					strArg := '');
				eMotionState := WAIT_FOR_TRIGGER;
			ELSE
				eMotionState := WAIT_FOR_NEW_VELOCITY; 
			END_IF
		END_IF
		
		
	WAIT_FOR_NEW_VELOCITY:
		IF nTargetVelocity <> nVelocityBuff THEN
			eMotionState := SET_LIMIT;
		ELSE
			bSetVelocity := FALSE;
			bBusy := FALSE; //FB 
		END_IF
		
	
	SET_LIMIT:
		bBusy := TRUE;
		nVelocityBuff := nTargetVelocity;
		IF nVelocityBuff < nVelocityLimitMin THEN
			bLimitActive := TRUE;
			nVelocityBuff := nVelocityLimitMin;
			nTargetVelocityAfterLimit := nVelocityLimitMin;
			ADSLOGSTR(msgCtrlMask := ADSLOG_MSGTYPE_HINT,
				msgFmtStr := 'Velocity exceeds limit: Minimum limit was set',
				strArg := '');
		ELSIF nVelocityBuff > nVelocityLimitMax THEN
			bLimitActive := TRUE;
			nVelocityBuff := nVelocityLimitMax;
			nTargetVelocityAfterLimit := nVelocityLimitMax;
			ADSLOGSTR(msgCtrlMask := ADSLOG_MSGTYPE_HINT,
				msgFmtStr := 'Velocity exceeds limit: Maximum limit was set',
				strArg := '');
		ELSE 
			bLimitActive := FALSE;
			nTargetVelocityAfterLimit := nTargetVelocity;
		END_IF
		nTargetVelocity := nVelocityBuff;
		eMotionState := SET_VELOCITY;
	
		
	SET_VELOCITY:
		//set velocity
		bWriteToFB := TRUE;
		fFlag(CLK := fbSetVelocity.bBusy); 		
		
		IF fbSetVelocity.bError THEN
			//Error when setting Target Velocity
			bSuccess := FALSE;
			bWriteToFB := FALSE;
			ADSLOGSTR(msgCtrlMask := ADSLOG_MSGTYPE_HINT,
				msgFmtStr := 'Error in set velocity',
				strArg := '');
			eMotionState := WAIT_FOR_TRIGGER;
		END_IF
		
		IF fFlag.Q THEN
			eMotionState := VALIDATE_VELOCITY;
		END_IF
		
		
	VALIDATE_VELOCITY:
		bGetStatusword := TRUE;
		fbGetStatusword(sNetId := sNetId,
			nSlaveAddr := nSlaveAddr,
			nIndex := 16#6041,
			nSubIndex := 0,
			pDstBuf := ADR(nStatusword),
			cbBufLen := SIZEOF(nStatusword),
			bExecute := bGetStatusword);
		fFlag(CLK := fbGetStatusword.bBusy);
		IF fFlag.Q THEN
			IF nStatusword.4 THEN
//				ADSLOGSTR(msgCtrlMask := ADSLOG_MSGTYPE_HINT,
//				msgFmtStr := 'Velocity is valid',
//				strArg := '');
			ELSE 
				bSuccess := FALSE;
				ADSLOGSTR(msgCtrlMask := ADSLOG_MSGTYPE_HINT,
					msgFmtStr := 'Error when validating velocity. Controlword not set.',
					strArg := '');
			END_IF
			fbGetStatusword(bExecute := FALSE);
			bSetVelocity := FALSE;
			bWriteToFB := FALSE;
			eMotionState := WAIT_FOR_NEW_VELOCITY;
		END_IF
		
END_CASE

METHOD GetVMaxLimit : BOOL
VAR_INPUT
END_VAR
fbGetVelocityLimitMax(sNetId := sNetID,
					nSlaveAddr := nSlaveAddr,
					nSubIndex := 2, //v_max
					nIndex := 16#6046, 
					pDstBuf := ADR(nVelocityLimitMax),
					cbBufLen := SIZEOF(nVelocityLimitMax),
					bExecute := TRUE);
fbGetVelocityLimitMax(bExecute := FALSE);
END_METHOD

METHOD GetVMinLimit : BOOL
VAR_INPUT
END_VAR
fbGetVelocityLimitMin(sNetId := sNetID,
					nSlaveAddr := nSlaveAddr,
					nSubIndex := 1, //v_min
					nIndex := 16#6046, 
					pDstBuf := ADR(nVelocityLimitMin),
					cbBufLen := SIZEOF(nVelocityLimitMin),
					bExecute := TRUE);
fbGetVelocityLimitMin(bExecute := FALSE);
END_METHOD

METHOD ReadLimits : BOOL
VAR_INPUT
END_VAR
fbReadVelocityLimits1(nSlaveAddr := GVL.nSlaveAddr,
			nIndex := 16#6046,
			nSubindex := 1, //v_min
			pDstBuf := ADR(nVelocityLimitMin),
			cbBufLen := SIZEOF(nVelocityLimitMin),
			bExecute := TRUE);
	
	fbReadVelocityLimits2(sNetId := GVL.sNetId,
			nSlaveAddr := GVL.nSlaveAddr,
			nIndex := 16#6046,
			nSubindex := 2, //v_max
			pDstBuf := ADR(nVelocityLimitMax),
			cbBufLen := SIZEOF(nVelocityLimitMax),
			bExecute := TRUE);
			
IF NOT fbReadVelocityLimits1.bBusy AND NOT fbReadVelocityLimits2.bBusy THEN
	fbReadVelocityLimits1(bExecute := FALSE); 
	fbReadVelocityLimits2(bExecute := FALSE); 
END_IF
END_METHOD

END_FUNCTION_BLOCK

// ---- POUs/ProfilePositionMode/FB_EnableDevice.TcPOU
FUNCTION_BLOCK FB_EnableDevice 
VAR_IN_OUT
	bTrigger			: BOOL;
END_VAR
VAR_INPUT
	sNetID				: T_AmsNetId;
	nSlaveAddr			: UINT;
END_VAR
VAR_OUTPUT
	bFinished			: BOOL;
	bSuccess			: BOOL;
END_VAR
VAR
	eState				: (WAIT_FOR_TRIGGER, SHUTDOWN, SWITCH_ON);
	tWait1				: TON;
	tWait2				: TON;
	fbGetStatusword		: FB_EcCoeSdoRead;
	nStatusword			: UINT;
	bGetStatusword		: BOOL;
	bExecuteTimer		: BOOL;
END_VAR

CASE eState OF
	WAIT_FOR_TRIGGER:
		IF bTrigger THEN
			bExecuteTimer	:= FALSE;
			bSuccess := TRUE;
			bFinished := FALSE;
			bTrigger := FALSE;
			eState := SHUTDOWN;
		END_IF
	
	SHUTDOWN:
		MAIN.Controlword.0 := 0;
		MAIN.Controlword.1 := 1;
		MAIN.Controlword.2 := 1;
		MAIN.Controlword.7 := 0;

		tWait1(PT := T#125MS,
			IN := bExecuteTimer);
			bExecuteTimer := TRUE;
		IF tWait1.Q THEN
			bExecuteTimer := FALSE;
			tWait2(IN := bGetStatusword,
				PT := T#250MS);
			fbGetStatusword(sNetId := sNetId,
				nSlaveAddr := nSlaveAddr,
				nIndex := 16#6041,
				nSubIndex := 0,
				pDstBuf := ADR(nStatusword),
				cbBufLen := SIZEOF(nStatusword),
				bExecute := bGetStatusword);
			bGetStatusword := TRUE;
			IF tWait2.Q THEN
				ADSLOGSTR(msgCtrlMask := ADSLOG_MSGTYPE_HINT,
					msgFmtStr := 'Shutdown',
					strArg := '');
				bExecuteTimer := FALSE;
				IF (nStatusword.0 = 1 AND nStatusword.5) 
					AND NOT (nStatusword.1 AND nStatusword.2 AND nStatusword.3
						AND nStatusword.6) THEN
 					eState := SWITCH_ON;
				ELSE 
					bSuccess := FALSE;
					bFinished := TRUE;
					eState := WAIT_FOR_TRIGGER;
				END_IF
			END_IF
		END_IF
		
	SWITCH_ON:
		ADSLOGSTR(msgCtrlMask := ADSLOG_MSGTYPE_HINT,
			msgFmtStr := 'Switch On',
			strArg := '');
		MAIN.Controlword.0 := 1;
		MAIN.Controlword.1 := 1;
		MAIN.Controlword.2 := 1;
		Main.Controlword.3 := 1;
		Main.Controlword.7 := 0;
		bExecuteTimer := TRUE;
		bGetStatusWord := TRUE;
		IF tWait1.Q THEN
			bExecuteTimer	:= FALSE;
			IF tWait2.Q THEN
				bGetStatusword := FALSE;
				IF nStatusword.0 AND nStatusword.1 AND nStatusword.5 
						AND NOT (nStatusword.2 AND nStatusword.3 AND nStatusword.6) THEN
					bSuccess := FALSE;
				END_IF
				bFinished := TRUE;
				eState := WAIT_FOR_TRIGGER;
			END_IF
		END_IF
END_CASE

END_FUNCTION_BLOCK

// ---- POUs/ProfilePositionMode/Motion.TcPOU
FUNCTION_BLOCK Motion
VAR_INPUT
	sNetID					: T_AmsNetId;
	nSlaveAddr				: UINT;
	nTargetPosition			: DINT;
END_VAR
VAR_OUTPUT
	bSuccess				: BOOL;
	bSetpointSet			: BOOL;
	bStartPositioning		: BOOL;
END_VAR
VAR_IN_OUT
//	aControlStatusWords		: ARRAY[1..2] OF INT; 			//0x6040 (Controlword), 0x6041 (Statusword)  
//	bTargetPosition			: BOOL;							//0x607A (Target Position)
	bMove					: BOOL;
END_VAR
VAR
	eMotionState			: (WAIT_FOR_TRIGGER, ENABLE_DEVICE, SET_SETPOINT, VALIDATE_SETPOINT, ACKNOWLEDGE_SET_POINT, WAIT_FOR_NEW_SETPOINT);
	fbEnableDevice			: FB_EnableDevice;
	fbSetSetpoint			: FB_EcCoeSdoWrite;
	fbGetStatusword			: FB_EcCoeSdoRead;
	tWait					: TON;
	tWait2					: TON;
	rTrig					: R_TRIG;
	nStatusword				: UINT;
	bGetStatusword			: BOOL;
	bExecuteWait			: BOOL;
	bSetSetpoint			: BOOL;
	nSetPointBuf			: DINT;
END_VAR

CASE eMotionState OF
	WAIT_FOR_TRIGGER:
		MAIN.Controlword := 0;
		bStartPositioning := FALSE;
		IF bMove THEN
			bSetpointSet := TRUE;
			bSuccess := TRUE;
			ADSLOGSTR(msgCtrlMask := ADSLOG_MSGTYPE_HINT,
				msgFmtStr := 'Enable Device',
				strArg := '');
			eMotionState := ENABLE_DEVICE;
		END_IF	

	ENABLE_DEVICE:
		fbEnableDevice (bTrigger := bMove,
						bSuccess => bSuccess,
						sNetId := sNetId,
						nSlaveAddr := nSlaveAddr);
		IF fbEnableDevice.bFinished THEN
			IF NOT bSuccess THEN
//				aControlStatusWords[1] := 0;
//				aControlStatusWords[2] := 0;
				ADSLOGSTR(msgCtrlMask := ADSLOG_MSGTYPE_HINT,
					msgFmtStr := 'Device not successfully enabled',
					strArg := '');
				eMotionState := WAIT_FOR_TRIGGER;
			ELSE
				ADSLOGSTR(msgCtrlMask := ADSLOG_MSGTYPE_HINT,
					msgFmtStr := 'Device successfully enabled',
					strArg := '');
				eMotionState := SET_SETPOINT;
			END_IF
		END_IF
		
	WAIT_FOR_NEW_SETPOINT:
		IF nTargetPosition <> nSetPointBuf THEN
			ADSLOGSTR(msgCtrlMask := ADSLOG_MSGTYPE_HINT,
				msgFmtStr := 'Set Setpoint',
				strArg := '');
				bStartPositioning := FALSE;
			eMotionState := SET_SETPOINT;
		END_IF
		
	SET_SETPOINT:
		bSetpointSet	:= TRUE;
		nSetPointBuf := nTargetPosition;
		fbSetSetpoint(sNetId := sNetID,
					nSlaveAddr := nSlaveAddr,
					nSubIndex := 0,
					nIndex := 16#607A,
					pSrcBuf := ADR(nTargetPosition),
					cbBufLen := SIZEOF(nTargetPosition),
					bExecute := bSetSetpoint);
		bSetSetpoint := TRUE;
		MAIN.TargetPosition := nTargetPosition;
		tWait(IN := bExecuteWait,
				PT := T#175MS); 
		bExecuteWait := TRUE;
		IF tWait.Q THEN
			bExecuteWait := FALSE;
			IF fbSetSetpoint.bError THEN
				//Error when setting Target Position
				bSuccess := FALSE;
				bSetSetpoint := FALSE;
				eMotionState := WAIT_FOR_TRIGGER;
			ELSE
				ADSLOGSTR(msgCtrlMask := ADSLOG_MSGTYPE_HINT,
					msgFmtStr := 'Validate Setpoint',
					strArg := '');
				eMotionState := VALIDATE_SETPOINT;
			END_IF
		END_IF
 
	VALIDATE_SETPOINT:
		bExecuteWait := TRUE;
		MAIN.Controlword.4 := 1;
		fbGetStatusword(sNetId := sNetId,
			nSlaveAddr := nSlaveAddr,
			nIndex := 16#6041,
			nSubIndex := 0,
			pDstBuf := ADR(nStatusword),
			cbBufLen := SIZEOF(nStatusword),
			bExecute := bGetStatusword);
		IF tWait.Q THEN
			bExecuteWait := FALSE;
			tWait2(IN := bGetStatusword,
				PT := T#250MS);
			bGetStatusword := TRUE;
			IF tWait2.Q THEN
				bGetStatusword := FALSE;
				IF nStatusword.12 THEN
					eMotionState := ACKNOWLEDGE_SET_POINT;
				ELSE 
					bSetSetpoint := FALSE;
					bSuccess := FALSE;
//					aControlStatusWords[1] := 0;
//					aControlStatusWords[2] := 0;
					ADSLOGSTR(msgCtrlMask := ADSLOG_MSGTYPE_HINT,
						msgFmtStr := 'Error when validating setpoint',
						strArg := '');
					eMotionState := WAIT_FOR_TRIGGER;
				END_IF
			END_IF
		END_IF
		
	ACKNOWLEDGE_SET_POINT:
		ADSLOGSTR(msgCtrlMask := ADSLOG_MSGTYPE_HINT,
			msgFmtStr := 'Acknowledge Setpoint',
			strArg := '');
		bGetStatusword := TRUE;
		IF tWait2.Q AND nStatusword.12 THEN
			bStartPositioning := TRUE;
			bGetStatusword := FALSE;
			//Set point acknowledge is set back
			MAIN.Controlword.4 := 0;
			ADSLOGSTR(msgCtrlMask := ADSLOG_MSGTYPE_HINT,
				msgFmtStr := 'Wait for new Setpoint',
				strArg := '');
			eMotionState := WAIT_FOR_NEW_SETPOINT;
		ELSE
			//TODO FAULT
			eMotionState := WAIT_FOR_TRIGGER;
		END_IF
END_CASE

END_FUNCTION_BLOCK

// ---- POUs/P_ProfilePositionModeTest.TcPOU
PROGRAM P_ProfilePositionModeTest
VAR
	fbMoveInProfilePosition				: Motion;
	fbGetCurrentPosition				: FB_EcCoeSdoRead;
	fbGetStatusword						: FB_EcCoeSdoRead;
	fbGetPositionWindow					: FB_EcCoeSdoRead;
	fbGetPositionDemandValue			: FB_EcCoeSdoRead;
	fbGetMinPositionRangeLimit			: FB_EcCoeSdoRead;
	fbGetMaxPositionRangeLimit			: FB_EcCoeSdoRead;
	tGetCurrentPosition					: TON;
	ftGetStatusword						: F_TRIG;
	ftGetPositionDemandValue			: F_TRIG;
	ftGetPositionRangeLimit				: F_TRIG;
	bGetCurrentPosition					: BOOL;
	bMove								: BOOL; 
	bExecuteTimer						: BOOL;
	bGetStatusword						: BOOL;
	bGetParameters						: BOOL;
	bSetPositioningOptionCode			: BOOL;
	bGetPositionDemandValue				: BOOL;
	bBasicOperationAbsStarted			: BOOL;
	bBasicOperationAbsFinished			: BOOL := FALSE;
	bPositioningOptionCodeSet			: BOOL;
	bTargetReached						: BOOL;
	bTestAbsolutePositioning			: BOOL;
	nTargetPosition						: DINT;
	nCurrentPosition					: DINT;
	nTargetPositionBuf					: DINT;  
	nPositionDemandValue				: DINT;
	nStatusword							: UINT;
	nPositionWindow						: UDINT;
	
	
	bTest								: BOOL;
	bAusprobieren						: BOOL;
END_VAR

VAR
	bBasicOperationAbs					: BOOL;
	bBasicOperationRel					: BOOL;
	bPositioningOptionCode				: BOOL;
END_VAR

//For Test Set of Setpoints
VAR
	bSetOfSetpointFinished 				: BOOL;
	nCurrentPositionBuf					: DINT;
	bSetpointSet						: BOOL;  //For both -> Test Change Immediately
	bSetOfSetpoints						: BOOL;
	bStartBasicOperationAbs				: BOOL;
	bTestSetOfSetpoints					: BOOL;
	bSetOfSetpointsFinished				: BOOL;
END_VAR

//Fo Test Change Immediately
VAR
	bTestChangeImmediately				: BOOL;
	bChangeImmediatelyFinished			: BOOL;
	bChangeImmediately					: BOOL;
END_VAR

//For test of relative Positioninig
VAR
	ftSetPositioningOptionCode			: F_TRIG;
	fbSetPositioningOptionCode			: FB_EcCoeSdoWrite;
	bTestRelativePositioning			: BOOL;
	bRelativePositioning				: BOOL := TRUE;
	bTestRelativePositioningFinished		: BOOL;
	bRelativePositioningFinished		: BOOL;
	nPositioningOptionCode				: DINT;
	nCounter							: DINT;
END_VAR

VAR
	bTestSupportedPPObjects				: BOOL;
	eTestSupportedPPObjects				: (POSITION_RANGE_LIMIT, SOFTWARE_POSITION_LIMIT, MAX_PROFILE_VELOCITY,
											MAX_MOTOR_SPEED, PROFILE_VELOCITY, END_VELOCITY, PROFILE_ACCELERATION,
											PROFILE_DECELERATION, MOTION_PROFILE_TYPE, MAX_ACCELERATION, MAX_DECELERATION);
	ePositionRangeLimitState			: (GET_CURRENT_POSITION_RANGE_LIMIT, SET_POSITION_RANGE_LIMIT, 
											TEST_POSITION_LIMIT, RESET_POSITION_RANGE_LIMIT); 
	eSoftwarePositionLimitState			: (GET_CURRENT_SOFTWARE_LIMITS, SET_SOFTWARE_LIMITS, 
											TEST_SOFTWARE_LIMITS, RESET_SOFTWARE_LIMITS);
	nMinPositionRangeLimit				: DINT;
	nMaxPositionRangeLimit				: DINT;
	nMinPositionRangeLimitTest			: DINT;
	nMaxPositionRangeLimitTest			: DINT;
	bGetPositionRangeLimit				: BOOL;
	bSetPositionRangeLimit				: BOOL;
	bPositionRangeLimit					: BOOL;
	bSoftwarePositionLimit				: BOOL;
	bMaxProfileVelocity					: BOOL;
	bMaxMotorSpeed						: BOOL;
	bProfileVelocity					: BOOL;
	bEndVelocity						: BOOL;
	bProfileAcceleration				: BOOL;
	bProfileDeceleration				: BOOL;
	bMotionProfileType					: BOOL;
	bMaxAcceleration					: BOOL;
	bMaxDeceleration					: BOOL;
	fbSetMinPositionRangeLimit			: FB_EcCoeSdoWrite;
	fbSetMaxPositionRangeLimit			: FB_EcCoeSdoWrite;
	fbGetMinSoftwarePositionRangeLimit	: FB_EcCoeSdoRead;
	fbGetMaxSoftwarePositionRangeLimit	: FB_EcCoeSdoRead;
	ftGetSoftwarePositionRangeLimit		: F_TRIG;
	ftSetPositionRangeLimit				: F_TRIG;
END_VAR

tGetCurrentPosition(IN := bGetCurrentPosition,
							PT := T#10MS);

ftGetStatusword(CLK := fbGetStatusword.bBusy);
ftGetPositionDemandValue(CLK := fbGetPositionDemandValue.bBusy);
ftGetPositionRangeLimit(CLK := fbGetMaxPositionRangeLimit.bBusy);
ftSetPositioningOptionCode(CLK := fbSetPositioningOptionCode.bBusy);

//TODO Position Range Limit		
							
IF tGetCurrentPosition.Q THEN
	bGetCurrentPosition := FALSE;
ELSE
	bGetCurrentPosition := TRUE;		
END_IF
fbMoveInProfilePosition(sNetID := GVL.sNetId,
						nSlaveAddr := GVL.nSlaveAddr,
						nTargetPosition := nTargetPosition,
						bMove := bMove);
fbGetStatusword(sNetId := GVL.sNetId,
				nSlaveAddr := GVL.nSlaveAddr,
				nIndex := 16#6041,
				nSubindex := 0,
				pDstBuf := ADR(nStatusWord),
				cbBufLen := SIZEOF(nStatusWord),
				bExecute := bGetStatusword);
fbGetCurrentPosition(sNetId := GVL.sNetId,
						nSlaveAddr := GVL.nSlaveAddr,
						nIndex := 16#6064,
						nSubIndex := 0,
						pDstBuf := ADR(nCurrentPosition),
						cbBufLen := SIZEOF(nCurrentPosition),
						bExecute := bGetCurrentPosition);
fbGetPositionWindow(sNetId := GVL.sNetId,
					nSlaveAddr := GVL.nSlaveAddr,
					nIndex := 16#6067,
					nSubIndex := 0,
					pDstBuf := ADR(nPositionWindow),
					cbBufLen := SIZEOF(nPositionWindow),
					bExecute := bGetParameters);
fbGetPositionDemandValue(sNetId := GVL.sNetId,
							nSlaveAddr := GVL.nSlaveAddr,
							nIndex := 16#60FC,
							nSubIndex := 0,
							pDstBuf := ADR(nPositionDemandValue),
							cbBufLen := SIZEOF(nPositionDemandValue),
							bExecute := bGetPositionDemandValue);
fbGetMinPositionRangeLimit(sNetId := GVL.sNetId,
							nSlaveAddr := GVL.nSlaveAddr,
							nSubIndex := 16#01,
							nIndex := 16#607B,
							pDstBuf := ADR(nMinPositionRangeLimit),
							cbBufLen := SIZEOF(nMinPositionRangeLimit),
							bExecute := bGetPositionRangeLimit);
fbGetMaxPositionRangeLimit(sNetId := GVL.sNetId,
							nSlaveAddr := GVL.nSlaveAddr,
							nSubIndex := 16#02,
							nIndex := 16#607B,
							pDstBuf := ADR(nMaxPositionRangeLimit),
							cbBufLen := SIZEOF(nMaxPositionRangeLimit),
							bExecute := bPositionRangeLimit);
							
fbSetPositioningOptionCode(sNetId := GVL.sNetId,
							nSlaveAddr := GVL.nSlaveAddr,
							nIndex := 16#60F2,
							nSubindex := 0,
							pSrcBuf := ADR(nPositioningOptionCode),
							cbBufLen := SIZEOF(nPositioningOptionCode),
							bExecute := bSetPositioningOptionCode);
fbSetMinPositionRangeLimit(sNetID := GVL.sNetId,
							nSlaveAddr := GVL.nSlaveAddr,
							nIndex := 16#607B,
							nSubindex := 16#01,
							pSrcBuf := ADR(nMinPositionRangeLimitTest),
							cbBufLen := SIZEOF(nMinPositionRangeLimitTest),
							bExecute := bSetPositionRangeLimit);
fbSetMaxPositionRangeLimit(sNetID := GVL.sNetId,
							nSlaveAddr := GVL.nSlaveAddr,
							nIndex := 16#607B,
							nSubindex := 16#02,
							pSrcBuf := ADR(nMaxPositionRangeLimitTest),
							cbBufLen := SIZEOF(nMaxPositionRangeLimitTest),
							bExecute := bSetPositionRangeLimit);
							
//TODO Position Range Limit
bGetParameters := TRUE;

IF bStartBasicOperationAbs THEN					
	//Basic Operation
	//Set-point is applied to the device
	//Move to absolute position is tested
	//Wait until Target reach Bit is set
	//Control if position is within error window
	
	//Target shall be an absolute value
	MAIN.Controlword.6 := 0;

	//Operation has not yet started and we are sure that initial position is obtained
	IF NOT bBasicOperationAbsStarted THEN
		nTargetPosition := nCurrentPosition + 5000000;
		//Start absolute positioning
		bMove := TRUE;	
		bBasicOperationAbsStarted := TRUE;
	END_IF
					
	//Target reached?
	bGetStatusword := TRUE;
	IF ftGetStatusword.Q THEN
		IF NOT nStatusword.10 THEN
			bGetStatusword := FALSE;
		ELSIF ((nCurrentPosition >= nTargetPosition - nPositionWindow)
				AND (nCurrentPosition <= nTargetPosition + nPositionWindow)) 
				AND fbMoveInProfilePosition.bStartPositioning THEN
			//absolute Positionining
			bBasicOperationAbs := TRUE;
			bBasicOperationAbsFinished := TRUE;
			bStartBasicOperationAbs := FALSE;
		ELSIF fbMoveInProfilePosition.bStartPositioning THEN
			bBasicOperationAbs := FALSE;
			bBasicOperationAbsFinished := TRUE;
			bStartBasicOperationAbs := FALSE;
		END_IF
		bGetStatusword := FALSE;
	END_IF
END_IF

//Test SetOfSetpoints
IF bTestSetOfSetpoints AND bBasicOperationAbsFinished AND NOT bSetOfSetpointsFinished THEN
	IF NOT bSetPointSet THEN
		MAIN.Controlword.5 := 0;
		nTargetPosition := nCurrentPosition + 100000000;
		nTargetPositionBuf := nTargetPosition;
		nCurrentPositionBuf := nCurrentPosition + 10000000/2;
		bSetPointSet := TRUE;
	END_IF
	IF (nCurrentPosition > nCurrentPositionBuf) AND bSetPointSet THEN
		nTargetPosition := nCurrentPositionBuf - 10000000/2;
	END_IF
	bSetOfSetpoints := TestChangeOfSetpoints(bActive => bSetOfSetpointsFinished);
	IF bSetOfSetpointsFinished THEN
		bSetPointSet := FALSE;
	END_IF
END_IF

//Change Immediately
IF bTestChangeImmediately AND bSetOfSetpointsFinished AND NOT bChangeImmediatelyFinished THEN
	IF NOT bSetPointSet THEN
		MAIN.Controlword.5 := 1;
		nTargetPosition := nCurrentPosition + 100000000;
		nTargetPositionBuf := nTargetPosition;
		nCurrentPositionBuf := nCurrentPosition + 10000000/2;
		bSetPointSet := TRUE;
	END_IF
	IF (nCurrentPosition > nCurrentPositionBuf) AND bSetPointSet THEN
		nTargetPosition := nCurrentPositionBuf - 10000000/2;
	END_IF
	bChangeImmediately := NOT TestChangeOfSetpoints(bActive => bChangeImmediatelyFinished);
END_IF

//Test relative positioning:
//Bit 6 of Controlword is set to 1

IF bTestRelativePositioning  AND bRelativePositioning THEN
	MAIN.Controlword.6 := 1;
	//positioning option code: 0
	//Positioning moves shall be performed relative to the preciding
	//target position
	IF nCounter = 0 AND NOT bSetpointSet THEN 
		SetPositioningOptionCode(nPositioningOptionCodeInput := 0);
		IF ftSetPositioningOptionCode.Q THEN
			bSetPositioningOptionCode := FALSE;
			nTargetPositionBuf := nCurrentPosition + 5000000;
			nTargetPosition := 5000000;
			bSetpointSet := TRUE;
			nCounter := nCounter + 1;
		END_IF
	END_IF

	//positioning option code: 2#0001
	//Positioning moves shall be performed relative to the actual
	//positioning demand value (16#60FC)
	IF nCounter = 1 AND NOT bSetpointSet THEN
		SetPositioningOptionCode(nPositioningOptionCodeInput := 2#0001);
		bGetPositionDemandValue := TRUE;
		IF ftGetPositionDemandValue.Q THEN
			bSetPositioningOptionCode := FALSE;
			nTargetPositionBuf := nPositionDemandValue + 6000000;
			nTargetPosition := 6000000;
			bSetpointSet := TRUE;
			nCounter := nCounter + 1;
		END_IF
	END_IF
	
	//positioning option code : 2#0010
	//Positioning moves shall be performed relative to the position
	//actual value (16#6064)
	IF nCounter = 2 AND NOT bSetpointSet THEN
		SetPositioningOptionCode(nPositioningOptionCodeInput := 2#0010);
		IF ftSetPositioningOptionCode.Q THEN
			bSetPositioningOptionCode := FALSE;
			nTargetPositionBuf := nCurrentPosition + 5000000;
			nTargetPosition := 5000000;
			bSetpointSet := TRUE;
			nCounter := nCounter + 1;
		END_IF
	END_IF
	
	bGetStatusword := TRUE;
	IF ftGetStatusword.Q THEN
		IF NOT nStatusword.10 THEN
			bGetStatusword := FALSE;
		ELSIF ((nCurrentPosition >= nTargetPositionBuf - nPositionWindow)
				AND (nCurrentPosition <= nTargetPositionBuf + nPositionWindow)) 
				AND bSetpointSet THEN
			//relative Positioning positive
			bTestRelativePositioning := TRUE;
			bSetpointSet := FALSE;
			IF nCounter = 3 THEN
				bTestRelativePositioning := FALSE;
				bTestRelativePositioningFinished := TRUE;
			END_IF
		ELSIF fbMoveInProfilePosition.bStartPositioning THEN
			bSetpointSet := FALSE;
			IF nCounter = 3 THEN
				bTestRelativePositioning := FALSE;
				//Actually redundant, but left in for consistensy reasons
				bTestRelativePositioningFinished := TRUE;
			END_IF
		END_IF
		bGetStatusword := FALSE;
	END_IF
END_IF

IF bTestSupportedPPObjects AND bTestRelativePositioningFinished THEN
	//607A - Target Position mode - already tested
	CASE eTestSupportedPPObjects OF
		//607B Position range limit
		//Object indicates maximum and minimum position range limit. It shall limit the range of the input value
		//On reaching or exeeding these limits, the input value shall wrap automatically to the other end of range
		POSITION_RANGE_LIMIT:
			CASE ePositionRangeLimitState OF
				GET_CURRENT_POSITION_RANGE_LIMIT:
					bGetPositionRangeLimit := TRUE;
					IF ftGetPositionRangeLimit.Q THEN
						ePositionRangeLimitState := SET_POSITION_RANGE_LIMIT;
					END_IF
					
				SET_POSITION_RANGE_LIMIT:
					nMinPositionRangeLimitTest := 1000000;
					nMaxPositionRangeLimitTest := nCurrentPosition + 5000000/2;
					bSetPositionRangeLimit := TRUE;
					IF ftSetPositionRangeLimit.Q THEN
						bSetPositionRangeLimit := FALSE;
						nTargetPosition := 5000000;
						ePositionRangeLimitState := TEST_POSITION_LIMIT;
					END_IF
					
				TEST_POSITION_LIMIT:
					bGetStatusword := TRUE;
					IF ftGetStatusword.Q THEN
						IF NOT nStatusword.10 THEN
							bGetStatusword := FALSE;
						ELSIF ((nCurrentPosition >=  (nMinPositionRangeLimitTest + 5000000/2) - nPositionWindow)
							AND (nCurrentPosition <= (nMinPositionRangeLimitTest + 5000000/2) + nPositionWindow)) 
							AND fbMoveInProfilePosition.bStartPositioning THEN
							bPositionRangeLimit := TRUE;
							ePositionRangeLimitState := RESET_POSITION_RANGE_LIMIT;
						ELSIF fbMoveInProfilePosition.bStartPositioning THEN
							bPositionRangeLimit := FALSE;
							ePositionRangeLimitState := RESET_POSITION_RANGE_LIMIT;
						END_IF
						bGetStatusword := FALSE;
					END_IF
				
				RESET_POSITION_RANGE_LIMIT:
					nMinPositionRangeLimitTest := nMinPositionRangeLimit;
					nMaxPositionRangeLimitTest := nMaxPositionRangeLimit;
					bSetPositionRangeLimit := TRUE;
					IF ftSetPositionRangeLimit.Q THEN
						eTestSupportedPPObjects := SOFTWARE_POSITION_LIMIT;
					END_IF	
			END_CASE

		//607D Software position limit
		SOFTWARE_POSITION_LIMIT:
			
				ePositionRangeLimitState := GET_CURRENT_POSITION_RANGE_LIMIT;
			
			

//607F Max profile velocity

//6080 Max motor speed

//6081 Profile velocity

//6082 End velocity

//6083 Profile acceleration

//6084 Profile deceleration 

//6085 Quick stop deceleration
//-> to be tested during quick stop tests

//6086 Motion profile type

//60C5 Max acceleration

//60C6 Max deceleration
	END_CASE
END_IF

METHOD SetPositioningOptionCode 
VAR_INPUT
	nPositioningOptionCodeInput		: DINT;
END_VAR
nPositioningOptionCode := nPositioningOptionCodeInput;
bSetPositioningOptionCode := TRUE;
END_METHOD

METHOD TestChangeOfSetpoints : BOOL
VAR_OUTPUT
	bActive		: BOOL;
END_VAR
IF ((nCurrentPosition >= nTargetPositionBuf - nPositionWindow)
	AND (nCurrentPosition <= nTargetPositionBuf + nPositionWindow)) THEN
	bActive := TRUE;
	bSetOfSetPointsFinished := TRUE;
ELSIF ((nCurrentPosition >= nTargetPosition - nPositionWindow)
	AND (nCurrentPosition <= nTargetPosition + nPositionWindow)) THEN
	TestChangeOfSetpoints := FALSE;
	bActive := TRUE;
END_IF
END_METHOD

END_PROGRAM

// ---- POUs/StartUpTests.TcPOU
PROGRAM StartUpTests
VAR CONSTANT
	stPlcErrorInit			: ST_PlcErrorStartUp := (bPlcError := FALSE, bErrorCode := [0,0,0,0]);
END_VAR

VAR
	eStartUpState 			: (WAIT_FOR_TRIGGER, TEST_SWITCH_ON_DISABLED, 
								SET_MODE_OF_OPERATION, TEST_MODE_OF_OPERATION, GET_TEMPERATURE, CHECK_PLC_ERROR);
	fbSetModeOfOperation	: FB_EcCoeSdoWrite;
	fbGetModeOfOperation	: FB_EcCoeSdoRead;
	fbGetDriveTemperature	: FB_EcCoeSdoRead;
	fbGetMotorTemperature	: FB_EcCoeSdoRead;
	stPlcError				: ST_PlcErrorStartUp;
	tTimeout				: TON;
	tWait1					: TON;
	tWait2					: TON;
	tWait					: TON;
	counter					: INT := -1;
	modeOfOperation			: INT;
	bExecuteChangeMOP		: BOOL;	
	bTestChangeMOP			: BOOL;
END_VAR
VAR_IN_OUT
	bTrigger				: BOOL;
	aTemperatureObjects		: ARRAY[1..2] OF INT;
	aMOPObjects				: ARRAY[1..2] OF INT;
	aControlStatusWords		: ARRAY[1..2] OF INT;
END_VAR
VAR_OUTPUT
	bSwitchOnDisabled		: BOOL;
	bChangeModeOfOperation	: BOOL := TRUE;
	bFinished				: BOOL;
	nDriveTemperature		: INT;
	nMotorTemperature		: INT;
END_VAR
VAR_INPUT
	sNetID					: T_AmsNetId;
	nSlaveAddr				: UINT;
END_VAR

CASE eStartUpState OF
	WAIT_FOR_TRIGGER:
		IF bTrigger THEN
			bTrigger := FALSE;
			tTimeout.IN := FALSE;
			bSwitchOnDisabled := FALSE;
			bChangeModeOfOperation := FALSE;
			bFinished := FALSE;
			counter := 1;
			stPlcError := stPlcErrorInit;
			eStartUpState := TEST_SWITCH_ON_DISABLED;
		END_IF
	
	TEST_SWITCH_ON_DISABLED:
		tTimeout(IN := TRUE,
			PT := T#1000MS);
		IF MAIN.Statusword.6 THEN
			bSwitchOnDisabled := TRUE;
			eStartUpState := SET_MODE_OF_OPERATION;
		ELSIF tTimeout.Q THEN
			bSwitchOnDisabled := FALSE;
			aControlStatusWords[1] := 0;
			eStartUpState := SET_MODE_OF_OPERATION;
		END_IF
	
	SET_MODE_OF_OPERATION:
	bTestChangeMOP := FALSE;
		fbSetModeOfOperation(sNetId := sNetId,
							nSlaveAddr := nSlaveAddr,
							nSubIndex := 0,
							nIndex := 16#6060,
							pSrcBuf := ADR(counter),
							cbBufLen := SIZEOF(counter),
							bExecute := bExecuteChangeMOP);
		tWait1(PT := T#2S, 
			IN := bExecuteChangeMOP);
		bExecuteChangeMOP := TRUE;				
		IF tWait1.Q THEN
			eStartUpState := TEST_MODE_OF_OPERATION;
		END_IF

	TEST_MODE_OF_OPERATION:
		bExecuteChangeMOP := FALSE;	
		fbGetModeOfOperation(sNetId := sNetId,
							nSlaveAddr := nSlaveAddr,
							nSubIndex := 0,
							nIndex := 16#6061,
							pDstBuf := ADR(modeOfOperation),
							cbBufLen := SIZEOF(modeOfOperation),
							bExecute := bTestChangeMOP);
		tWait2(PT := T#2S,
				IN := bTestChangeMOP);
		bTestChangeMOP := TRUE; 
		IF tWait2.Q THEN
			IF NOT modeOfOperation = counter AND counter <> 5 THEN
				bChangeModeOfOperation := FALSE;
				aMOPObjects[1] := 0;
				aMOPObjects[2] := 0;
			END_IF
			counter := counter + 1;
			IF counter < 11 THEN
				eStartUpState := SET_MODE_OF_OPERATION;
			ELSE
				eStartUpState := GET_TEMPERATURE;
			END_IF
		END_IF
	
	GET_TEMPERATURE:
		fbGetDriveTemperature(sNetId := sNetId,
							nSlaveAddr := nSlaveAddr,
							nSubIndex := 0,
							nIndex := 16#2200,
							pDstBuf := ADR(nDriveTemperature),
							cbBufLen := SIZEOF(nDriveTemperature),
							bExecute := TRUE);
		fbGetMotorTemperature(sNetId := sNetId,
							nSlaveAddr := nSlaveAddr,
							nSubIndex := 0,
							nIndex := 16#2202,
							pDstBuf := ADR(nMotorTemperature),
							bExecute := TRUE);							
		tWait(IN := TRUE,
			PT := T#125MS);
		IF tWait.Q THEN
			tWait.IN := FALSE;
		//	eStartUpState := CHECK_PLC_ERROR;
		END_IF
		
		CHECK_PLC_ERROR:
			IF fbSetModeOfOperation.bError OR fbGetModeOfOperation.bError OR
				fbGetDriveTemperature.bError OR fbGetMotorTemperature.bError THEN
				stPlcError.bPlcError := TRUE;
				IF fbSetModeOfOperation.bError THEN
					stPlcError.bErrorCode[1] := fbSetModeOfOperation.nErrId;
					aMOPObjects[1] := 0;
				END_IF
				IF fbGetModeOfOperation.bError THEN
					stPlcError.bErrorCode[2] := fbGetModeOfOperation.nErrId;
					aMOPObjects[2] := 0;		
				END_IF
				IF fbGetDriveTemperature.bError THEN
					stPlcError.bErrorCode[3] := fbGetDriveTemperature.nErrId;
					aTemperatureObjects[1] := 0;
				END_IF
				IF fbGetMotorTemperature.bError THEN
					stPlcError.bErrorCode[4] := fbGetMotorTemperature.nErrId;
					aTemperatureObjects[2] := 0;
				END_IF
			END_IF
			bFinished := TRUE;
			eStartUpState := WAIT_FOR_TRIGGER;
END_CASE

END_PROGRAM
